FUNCTION_BLOCK EV_COUNTER
  (* Standard: 61499-2 *)
  (* Version 0.0, 2002-12-16, HDF, Schneider Automation *)
  (* Compiler header: package fb.rt.ita; *)
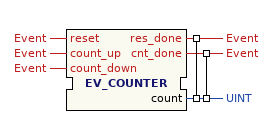
  EVENT_INPUT
    reset;
    count_up;
    count_down;
  END_EVENT
  EVENT_OUTPUT
    res_done WITH count;
    cnt_done WITH count;
  END_EVENT
  VAR_OUTPUT
    count : UINT;
  END_VAR
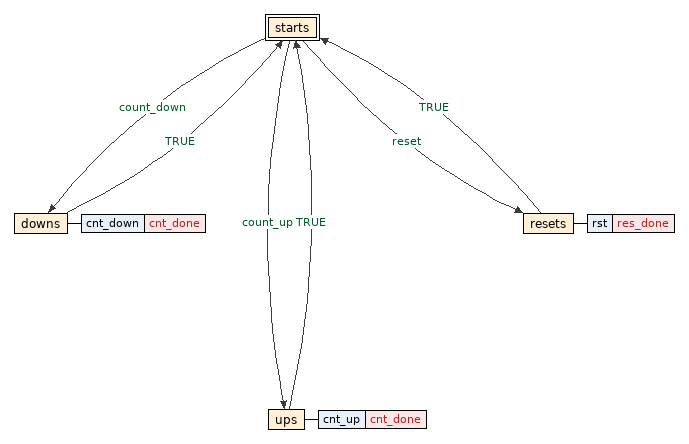
  EC_STATES
    starts;
    resets : rst -> res_done;
    ups : cnt_up -> cnt_done;
    downs : cnt_down -> cnt_done;
  END_STATES
  EC_TRANSITIONS
    starts TO resets := reset;
    starts TO ups := count_up;
    starts TO downs := count_down;
    resets TO starts := TRUE;
    ups TO starts := TRUE;
    downs TO starts := TRUE;
  END_TRANSITIONS
  ALGORITHM rst IN ST:
count:=0;
  END_ALGORITHM
  ALGORITHM cnt_up IN ST:
count:=count+1;
  END_ALGORITHM
  ALGORITHM cnt_down IN ST:
count:=count-1;
  END_ALGORITHM
END_FUNCTION_BLOCK
